{attribute addProperty BoxType "EK1122-0000-0018"}
{attribute addProperty Id "Beckhoff_EP6xxxsub_EK1100EK1100_179A0949162A_0001_EP6001_0002_0020EP6001_7904467646658.25A_0002_EP6001_0002_0021EP6001_7904467646658.25A_0003_EP6002_0002_0016EP6002_1BCFC91E850106.25A_0004_EP6002_0002_0017EP6002_320F021A850106.25A_0005_EP6002_0002_0018EP6002_320F021A850106.25A_0006_EP6002_0002_0019EP6002_320F021A850106.25A_0007_EP6002_0002_0020EP6002_320F021A850106.25A_0008_EP6002_0002_0021EP6002_320F021A850106.25A_0009_EP6002_0002_0023EP6002_FC20A988850106.25A_0010_EP6002_0002_0024EP6002_FC20A988850106.25A_0011_EP6090_0000_0017EP6090_7D66C95013016.25A_0012_EP6224_0002_0016EP6224_69FFDAE721026.25A_0013_EP6224_0042_0016EP6224_6FAF51E924230.25A_0014_EP6224_2022_0016EP6224_FF3BC86C17822.25A_0015_EP6224_2022_0017EP6224_FF3BC86C17822.25A_0016_EP6224_2022_0018EP6224_3990B4B417822.25A_0017_EP6224_3022_0016EP6224_FF3BC86C17822.25A_0018_EP6224_3022_0017EP6224_3990B4B417822.25A_0019_EP6228_0022_0016EP6228_B7929BD921026.25A_0020_EP6228_0022_0017EP6228_B7929BD921026.25A_0021_EP6228_0022_0018EP6228_B7929BD921026.25A_0022_EP6228_0042_0016EP6228_E048681B27434.25A_0023_EP6228_3032_0016EP6228_B7929BD921026.25A_0024_EP6228_3132_0016EP6228_ABD94E9E24230.25A_0025_EP6228_3142_0016EP6228_ABD94E9E24230.25A_0026_EP6601_0002_0018EP6601_194A340D8010"}
{attribute addProperty CRC "3886009613"}
{attribute addProperty SizeInBites "10898"}
{attribute addProperty SizeInBytes "1362.25"}
TYPE Beckhoff_EP6xxxEK1122_E79FCD0D EXTENDS EK1122_179A0949 :
STRUCT
	{attribute addProperty Name "Beckhoff_EP6xxxsub_EK1100"}
	Beckhoff_EP6xxxsub_EK1100 : EK1100_179A0949;
	{attribute addProperty Name "A_0001_EP6001_0002_0020"}
	A_0001_EP6001_0002_0020 : EP6001_79044676;
	{attribute addProperty Name "A_0002_EP6001_0002_0021"}
	A_0002_EP6001_0002_0021 : EP6001_79044676;
	{attribute addProperty Name "A_0003_EP6002_0002_0016"}
	A_0003_EP6002_0002_0016 : EP6002_1BCFC91E;
	{attribute addProperty Name "A_0004_EP6002_0002_0017"}
	A_0004_EP6002_0002_0017 : EP6002_320F021A;
	{attribute addProperty Name "A_0005_EP6002_0002_0018"}
	A_0005_EP6002_0002_0018 : EP6002_320F021A;
	{attribute addProperty Name "A_0006_EP6002_0002_0019"}
	A_0006_EP6002_0002_0019 : EP6002_320F021A;
	{attribute addProperty Name "A_0007_EP6002_0002_0020"}
	A_0007_EP6002_0002_0020 : EP6002_320F021A;
	{attribute addProperty Name "A_0008_EP6002_0002_0021"}
	A_0008_EP6002_0002_0021 : EP6002_320F021A;
	{attribute addProperty Name "A_0009_EP6002_0002_0023"}
	A_0009_EP6002_0002_0023 : EP6002_FC20A988;
	{attribute addProperty Name "A_0010_EP6002_0002_0024"}
	A_0010_EP6002_0002_0024 : EP6002_FC20A988;
	{attribute addProperty Name "A_0011_EP6090_0000_0017"}
	A_0011_EP6090_0000_0017 : EP6090_7D66C950;
	{attribute addProperty Name "A_0012_EP6224_0002_0016"}
	A_0012_EP6224_0002_0016 : EP6224_69FFDAE7;
	{attribute addProperty Name "A_0013_EP6224_0042_0016"}
	A_0013_EP6224_0042_0016 : EP6224_6FAF51E9;
	{attribute addProperty Name "A_0014_EP6224_2022_0016"}
	A_0014_EP6224_2022_0016 : EP6224_FF3BC86C;
	{attribute addProperty Name "A_0015_EP6224_2022_0017"}
	A_0015_EP6224_2022_0017 : EP6224_FF3BC86C;
	{attribute addProperty Name "A_0016_EP6224_2022_0018"}
	A_0016_EP6224_2022_0018 : EP6224_3990B4B4;
	{attribute addProperty Name "A_0017_EP6224_3022_0016"}
	A_0017_EP6224_3022_0016 : EP6224_FF3BC86C;
	{attribute addProperty Name "A_0018_EP6224_3022_0017"}
	A_0018_EP6224_3022_0017 : EP6224_3990B4B4;
	{attribute addProperty Name "A_0019_EP6228_0022_0016"}
	A_0019_EP6228_0022_0016 : EP6228_B7929BD9;
	{attribute addProperty Name "A_0020_EP6228_0022_0017"}
	A_0020_EP6228_0022_0017 : EP6228_B7929BD9;
	{attribute addProperty Name "A_0021_EP6228_0022_0018"}
	A_0021_EP6228_0022_0018 : EP6228_B7929BD9;
	{attribute addProperty Name "A_0022_EP6228_0042_0016"}
	A_0022_EP6228_0042_0016 : EP6228_E048681B;
	{attribute addProperty Name "A_0023_EP6228_3032_0016"}
	A_0023_EP6228_3032_0016 : EP6228_B7929BD9;
	{attribute addProperty Name "A_0024_EP6228_3132_0016"}
	A_0024_EP6228_3132_0016 : EP6228_ABD94E9E;
	{attribute addProperty Name "A_0025_EP6228_3142_0016"}
	A_0025_EP6228_3142_0016 : EP6228_ABD94E9E;
	{attribute addProperty Name "A_0026_EP6601_0002_0018"}
	A_0026_EP6601_0002_0018 : EP6601_194A340D;
END_STRUCT
END_TYPE

(* stored: Version 1.2.0.0, ProductVersion 3.1.4024.9
   DUT Beckhoff_EP6xxxEK1122_E79FCD0D: Id {060a71db-8b00-430d-8f6b-ccb545dc07e8} *)
